FUNCTION HLI3_GetVEChannelDIntValue : DINT
VAR_INPUT
	/// HLI Channel Index 
	nChanIdx: INT;
	/// Index of variable  range 1 ...     HLI_VE_VALUEMAX 
	nVEIndex: DINT;
	/// Array index. 0 if no array 
	nArrayIndex: DINT := 0;
	/// serves acess to the global variable array 
	bGlobal: BOOL;
END_VAR
VAR
	pVeData: POINTER TO VEData := 0;
	/// Size of the datatype of the returned value 
	iDatatypeSize: DINT;
	ptr: POINTER TO DINT;
	ChIdx: UDINT;
	SizeField: DINT := 0;
END_VAR

(* ========================================================= *)
(*    FUN: GetVEChannelDINTValue                            *)
(* --------------------------------------------------------- *)
(*   Desc: Reads a V.E.Variable of DINT                    *)
(* 	 Author: CL  / TV                                        *)
(*   Date: 16.05.2006                                        *)
(*   Last: 28.01.2013                                        *)
(*   Rev.: 1.3                                               *)
(* ========================================================= *)

IF  nVEIndex >= 0 AND
	nArrayIndex >= 0 THEN

	(* test if channel specific or global *)
	IF bGlobal = FALSE  THEN
		IF NOT HLI3_CheckChannelValid(nChannel := nChanIdx) THEN
			RETURN;
		END_IF
				
		pVeData := gpVECh[nChanIdx];
	ELSE
		pVeData := gpVEGlobal;
	END_IF

	IF pVeData <> 0 THEN
		IF pVeData <> 0 THEN
			iDatatypeSize := SIZEOF(ptr^);
                         	ptr := pVeData +  24  * nVEIndex + (iDatatypeSize * nArrayIndex);
                           HLI3_GetVEChannelDIntValue := ptr^; (* successfully completed return *)
                END_IF
	END_IF
END_IF

END_FUNCTION

(* stored: Version 1.1.0.1, ProductVersion 3.1.4018.2
   POU HLI3_GetVEChannelDIntValue: Id {2de9f4ab-37c7-4bba-9822-8a3507e260c4}, SpecialFunc None *)
